FUNCTION HLI_ChannelSetSyntaxCheck : bool
VAR_INPUT
	nChan					: UDINT;			(* Number of channel *)
	nSyntaxCheck		: DINT;
END_VAR
VAR
	nHliChIdx			: UdINT;
END_VAR

(* ========================================================= *)
(*    FUN: HLI_ChannelSetSyntaxCheck                         *)
(* --------------------------------------------------------- *)
(*   Desc:                                                   *)
(* Author: MK                                                *)
(*   Date: 21.12.2011                                        *)
(*   Rev.: 1.0                                               *)
(* ========================================================= *)


nHliChIdx := nChan - 1;

IF nChan <= 0 OR gNrCh < nChan OR			(* check for channel no *)
	gpCh[nHliChIdx] = 0 THEN					(* check for zero pointer *)
	HLI_ChannelSetSyntaxCheck := FALSE;
	RETURN; (* e x i t *)
END_IF

gpCh[nHliChIdx]^.decoder_mc_control.execution_mode.command_w  := nSyntaxCheck;

HLI_ChannelSetSyntaxCheck := TRUE;

END_FUNCTION

(* stored: Version 1.1.0.1, ProductVersion 3.1.4018.5
   POU HLI_ChannelSetSyntaxCheck: Id {ed27d5b3-fe09-4f77-bcef-67f59cab96b7}, SpecialFunc None *)
